// TIA Portal project "HW_2000528_ST43_V18" (V18)

(* hardware
DEVICE "GSD device_5"  GSD.Device.PN
   slot 0: "wp4.3-dm262-l"  DataMan 260  DMR-260#-#0  5.5.0
      slot 0: "DataMan 260"  DataMan 260
      slot 1: "Interface"  Interface
         slot 1: "Port 1"  Port 1
   slot 0: "Rack"  Rack  V1.0
   slot 1: "Acquisition Control_1"  Acquisition Control
      slot 0: "Acquisition Control"  Acquisition Control
   slot 2: "Acquisition Status_1"  Acquisition Status
      slot 0: "Acquisition Status"  Acquisition Status
   slot 3: "Results Control_1"  Results Control
      slot 0: "Results Control"  Results Control
   slot 4: "Results Status_1"  Results Status
      slot 0: "Results Status"  Results Status
   slot 5: "Soft Event Control_1"  Soft Event Control
      slot 0: "Soft Event Control"  Soft Event Control
   slot 6: "User Data - 64 bytes_1"  User Data - 64 bytes
      slot 0: "User Data - 64 bytes"  User Data - 64 bytes
   slot 7: "Result Data - 64 bytes_1"  Result Data - 64 bytes
      slot 0: "Result Data - 64 bytes"  Result Data - 64 bytes
DEVICE "S71500/ET200MP station_2"  S7-1500 station
   slot 0: "Rail_0"  Rack  6ES7 590-1***0-0AA0
   slot 1: "PLC_4.3"  CPU 1515-2 PN  6ES7 515-2AM02-0AB0  V2.8
      slot 3: "CPU display_1"  6ES7591-1BA00-0AA0
      slot 32768: "PROFINET interface_1"  X1
         slot 32769: "Port_1"  X1 P1
         slot 32770: "Port_2"  X1 P2
      slot 33024: "PROFINET interface_2"  X2
         slot 33025: "Port_1"  X2 P1
      slot 34817: "Virtual CP interface port_1"  Virtual CP interface port  Virtual CP interface port
DEVICE "GSD device_4"  GSD.Device.PN
   slot 0: "CPX_ST43"  CPX Rev 30  TN 197330  V4.2.30
      slot 0: "CPX Rev 30"  CPX Rev 30
      slot 1: "PN-IO Interface"  PN-IO Interface
         slot 1: "Port 1"  Port 1
         slot 2: "Port 2"  Port 2
   slot 0: "Rack"  Rack  V1.0
   slot 1: "FB33 PNIO Module_1"  FB33 PNIO Module  TN 548755, CPX-FB33, Code F33
      slot 0: "FB33 PNIO Module"  FB33 PNIO Module
   slot 2: "MPA1S VMPA1-FB-EMS-8 [8DO]_1"  MPA1S VMPA1-FB-EMS-8 [8DO]  TN 533360, VMPA1-FB-EMS-8, Code A
      slot 0: "MPA1S VMPA1-FB-EMS-8 [8DO]"  MPA1S VMPA1-FB-EMS-8 [8DO]
   slot 3: "MPA1G VMPA1-FB-EMG-8 [8DO]_1"  MPA1G VMPA1-FB-EMG-8 [8DO]  TN 533361, VMPA1-FB-EMG-8, Code AH
      slot 0: "MPA1G VMPA1-FB-EMG-8 [8DO]"  MPA1G VMPA1-FB-EMG-8 [8DO]
   slot 4: "MPA1G VMPA1-FB-EMG-8 [8DO]_2"  MPA1G VMPA1-FB-EMG-8 [8DO]  TN 533361, VMPA1-FB-EMG-8, Code AH
      slot 0: "MPA1G VMPA1-FB-EMG-8 [8DO]"  MPA1G VMPA1-FB-EMG-8 [8DO]
   slot 5: "MPA1G VMPA1-FB-EMG-8 [8DO]_3"  MPA1G VMPA1-FB-EMG-8 [8DO]  TN 533361, VMPA1-FB-EMG-8, Code AH
      slot 0: "MPA1G VMPA1-FB-EMG-8 [8DO]"  MPA1G VMPA1-FB-EMG-8 [8DO]
   slot 6: "MPA1G VMPA1-FB-EMG-8 [8DO]_4"  MPA1G VMPA1-FB-EMG-8 [8DO]  TN 533361, VMPA1-FB-EMG-8, Code AH
      slot 0: "MPA1G VMPA1-FB-EMG-8 [8DO]"  MPA1G VMPA1-FB-EMG-8 [8DO]
   slot 7: "MPA1G VMPA1-FB-EMG-8 [8DO]_5"  MPA1G VMPA1-FB-EMG-8 [8DO]  TN 533361, VMPA1-FB-EMG-8, Code AH
      slot 0: "MPA1G VMPA1-FB-EMG-8 [8DO]"  MPA1G VMPA1-FB-EMG-8 [8DO]
DEVICE "GSD device_1"  GSD.Device.PN
   slot 0: "wp4.3-dm262-r"  DataMan 260  DMR-260#-#0  5.5.0
      slot 0: "DataMan 260"  DataMan 260
      slot 1: "Interface"  Interface
         slot 1: "Port 1"  Port 1
   slot 0: "Rack"  Rack  V1.0
   slot 1: "Acquisition Control_1"  Acquisition Control
      slot 0: "Acquisition Control"  Acquisition Control
   slot 2: "Acquisition Status_1"  Acquisition Status
      slot 0: "Acquisition Status"  Acquisition Status
   slot 3: "Results Control_1"  Results Control
      slot 0: "Results Control"  Results Control
   slot 4: "Results Status_1"  Results Status
      slot 0: "Results Status"  Results Status
   slot 5: "Soft Event Control_1"  Soft Event Control
      slot 0: "Soft Event Control"  Soft Event Control
   slot 6: "User Data - 64 bytes_1"  User Data - 64 bytes
      slot 0: "User Data - 64 bytes"  User Data - 64 bytes
   slot 7: "Result Data - 64 bytes_1"  Result Data - 64 bytes
      slot 0: "Result Data - 64 bytes"  Result Data - 64 bytes
DEVICE "ET 200SP station_1"  ET 200SP-Station
   slot 0: "ET_200SP_ST43"  IM 155-6 PN ST  6ES7 155-6AU01-0BN0  V4.1
   slot 0: "Rack_0"  Rack  6ES5 710-8MAx1
   slot 1: "A3"  AI 4xU/I 2-wire ST  6ES7 134-6HD01-0BA1  V2.0
      slot 1: "A3"  AI 4xU/I 2-wire ST
   slot 2: "A4"  AI 4xU/I 2-wire ST  6ES7 134-6HD01-0BA1  V2.0
      slot 1: "A4"  AI 4xU/I 2-wire ST
   slot 3: "A5"  AI 4xU/I 2-wire ST  6ES7 134-6HD01-0BA1  V2.0
      slot 1: "A5"  AI 4xU/I 2-wire ST
   slot 4: "DI 16x24VDC ST_1"  DI 16x24VDC ST  6ES7 131-6BH01-0BA0  V0.0
      slot 1: "DI 16x24VDC ST_1"  DI 16x24VDC ST
   slot 5: "DI 16x24VDC ST_2"  DI 16x24VDC ST  6ES7 131-6BH01-0BA0  V0.0
      slot 1: "DI 16x24VDC ST_2"  DI 16x24VDC ST
   slot 6: "DI 16x24VDC ST_3"  DI 16x24VDC ST  6ES7 131-6BH01-0BA0  V0.0
      slot 1: "DI 16x24VDC ST_3"  DI 16x24VDC ST
   slot 7: "DI 16x24VDC ST_4"  DI 16x24VDC ST  6ES7 131-6BH01-0BA0  V0.0
      slot 1: "DI 16x24VDC ST_4"  DI 16x24VDC ST
   slot 8: "DQ 16x24VDC/0.5A ST_1"  DQ 16x24VDC/0.5A ST  6ES7 132-6BH01-0BA0  V0.0
      slot 1: "DQ 16x24VDC/0.5A ST_1"  DQ 16x24VDC/0.5A ST
   slot 9: "DQ 16x24VDC/0.5A ST_2"  DQ 16x24VDC/0.5A ST  6ES7 132-6BH01-0BA0  V0.0
      slot 1: "DQ 16x24VDC/0.5A ST_2"  DQ 16x24VDC/0.5A ST
   slot 10: "TM Pulse 2x24V_1"  TM Pulse 2x24V  6ES7 138-6DB00-0BB1  V1.0
      slot 1: "TM Pulse 2x24V_1"  TM Pulse 2x24V
   slot 11: "TM Pulse 2x24V_2"  TM Pulse 2x24V  6ES7 138-6DB00-0BB1  V1.0
      slot 1: "TM Pulse 2x24V_2"  TM Pulse 2x24V
   slot 12: "TM Pulse 2x24V_3"  TM Pulse 2x24V  6ES7 138-6DB00-0BB1  V1.0
      slot 1: "TM Pulse 2x24V_3"  TM Pulse 2x24V
   slot 13: "TM Pulse 2x24V_4"  TM Pulse 2x24V  6ES7 138-6DB00-0BB1  V1.0
      slot 1: "TM Pulse 2x24V_4"  TM Pulse 2x24V
   slot 14: "TM Pulse 2x24V_5"  TM Pulse 2x24V  6ES7 138-6DB00-0BB1  V1.0
      slot 1: "TM Pulse 2x24V_5"  TM Pulse 2x24V
   slot 15: "Server module_1"  Server module  6ES7 193-6PA00-0AA0  V1.1
      slot 1: "Server module_1"  Server module
   slot 127: "BA 2xRJ45"  BA 2xRJ45  6ES7 193-6AR00-0AA0  V0.0
      slot 1: "Port_1"  X1 P1 R  6ES7 193-6AR00-0AA0  V0.0
      slot 2: "Port_2"  X1 P2 R  6ES7 193-6AR00-0AA0  V0.0
*)

// ===== PLC "PLC_4.3"  CPU 1515-2 PN =====

VAR_GLOBAL   // PLC tag table "Default tag table"
   "Clock_Byte" AT %MB0 : Byte;
   "Clock_10Hz" AT %M0.0 : Bool;
   "Clock_5Hz" AT %M0.1 : Bool;
   "Clock_2.5Hz" AT %M0.2 : Bool;
   "Clock_2Hz" AT %M0.3 : Bool;
   "Clock_1.25Hz" AT %M0.4 : Bool;
   "Clock_1Hz" AT %M0.5 : Bool;
   "Clock_0.625Hz" AT %M0.6 : Bool;
   "Clock_0.5Hz" AT %M0.7 : Bool;
   "System_Byte" AT %MB1 : Byte;
   "FirstScan" AT %M1.0 : Bool;
   "DiagStatusUpdate" AT %M1.1 : Bool;
   "AlwaysTRUE" AT %M1.2 : Bool;
   "AlwaysFALSE" AT %M1.3 : Bool;
END_VAR

ORGANIZATION_BLOCK "Main"   // OB1, LAD, ProgramCycle
TITLE = "Main Program Sweep (Cycle)"
{ S7_Optimized_Access := 'TRUE' }
VERSION : 0.1
   VAR_INPUT
      Initial_Call : Bool;   // Initial call of this OB
      Remanence : Bool;   // =True, if remanent data are available
   END_VAR
BEGIN
END_ORGANIZATION_BLOCK